FUNCTION_BLOCK Gripper1Ctrl (* Basic Function Block Type *)
  (* Standard: 61499-2 *)
  (* Version 0.0, 3/23/2016, Aalto_IT, nxtControl GmbH, Template *)
  PACKAGE Main;
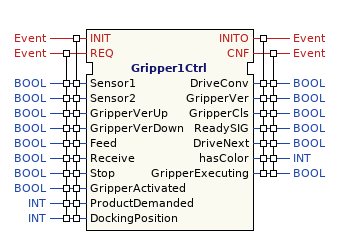
  EVENT_INPUT
    INIT WITH Sensor1, Sensor2, GripperVerUp, GripperVerDown, Feed, Receive, Stop, GripperActivated, ProductDemanded, DockingPosition; (* Initialization Request *)
    REQ WITH Sensor1, Sensor2, GripperVerUp, GripperVerDown, Feed, Receive, Stop, GripperActivated, ProductDemanded, DockingPosition; (* Normal Execution Request *)
  END_EVENT
  EVENT_OUTPUT
    INITO WITH DriveConv, GripperVer, GripperCls, ReadySIG, DriveNext, hasColor, GripperExecuting; (* Initialization Confirm *)
    CNF WITH DriveConv, GripperVer, GripperCls, ReadySIG, DriveNext, hasColor, GripperExecuting; (* Execution Confirmation *)
  END_EVENT
  VAR_INPUT
    Sensor1 : BOOL; (* Input event qualifier *)
    Sensor2 : BOOL;
    GripperVerUp : BOOL;
    GripperVerDown : BOOL;
    Feed : BOOL;
    Receive : BOOL;
    Stop : BOOL;
    GripperActivated : BOOL;
    ProductDemanded : INT;
    DockingPosition : INT;
  END_VAR
  VAR_OUTPUT
    DriveConv : BOOL; (* Output event qualifier *)
    GripperVer : BOOL;
    GripperCls : BOOL;
    ReadySIG : BOOL;
    DriveNext : BOOL;
    hasColor : INT;
    GripperExecuting : BOOL;
  END_VAR
  VAR
    TimeStamp : DATE_AND_TIME;
    SkipWorkCycle : BOOL;
  END_VAR
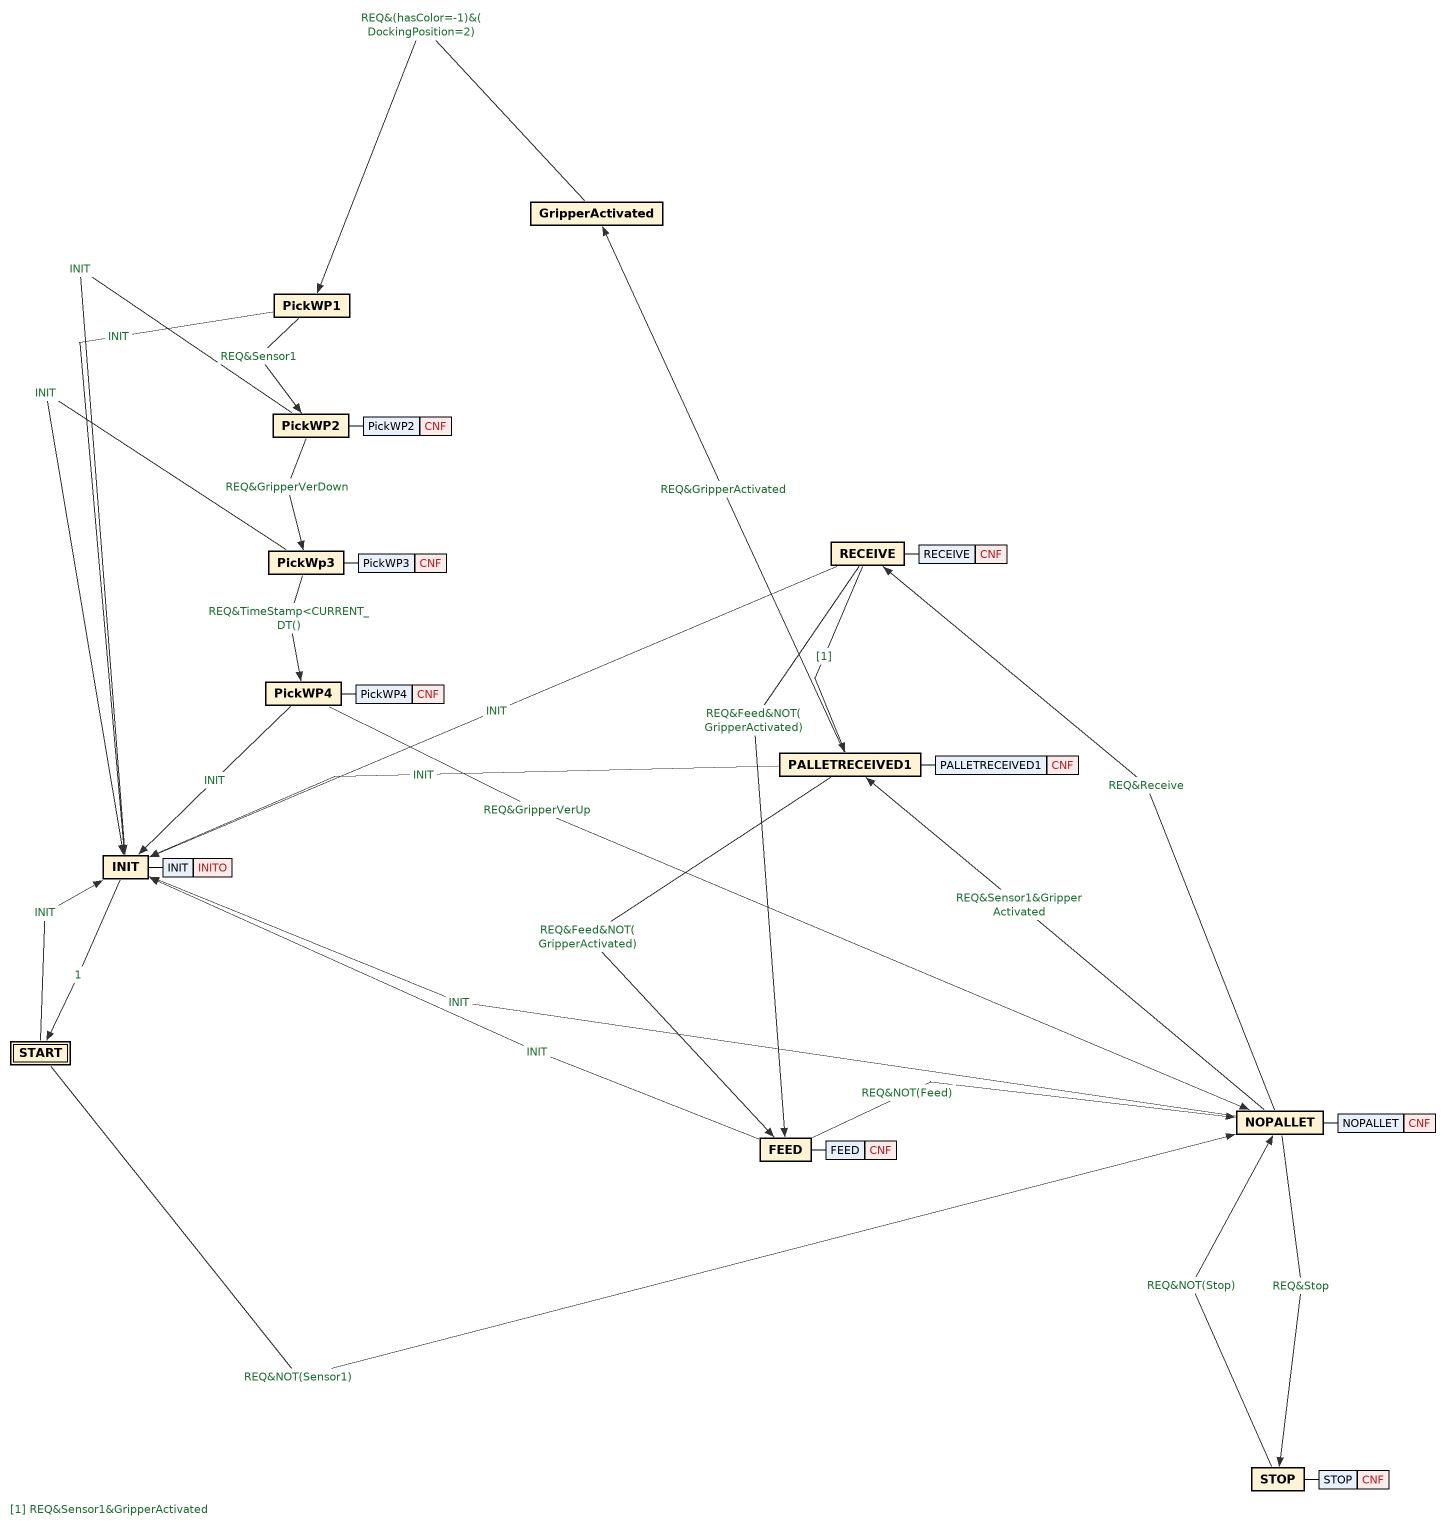
  EC_STATES
    START; (* Initial State *)
    INIT : INIT -> INITO; (* Initialization *)
    NOPALLET : NOPALLET -> CNF;
    PALLETRECEIVED1 : PALLETRECEIVED1 -> CNF;
    FEED : FEED -> CNF;
    RECEIVE : RECEIVE -> CNF;
    STOP : STOP -> CNF;
    GripperActivated;
    PickWP1;
    PickWP2 : PickWP2 -> CNF;
    PickWp3 : PickWP3 -> CNF;
    PickWP4 : PickWP4 -> CNF;
  END_STATES
  EC_TRANSITIONS
    START TO INIT := INIT;
    INIT TO START := 1;
    NOPALLET TO PALLETRECEIVED1 := REQ&Sensor1&GripperActivated;
    PALLETRECEIVED1 TO GripperActivated := REQ&GripperActivated;
    FEED TO NOPALLET := REQ&NOT(Feed);
    PALLETRECEIVED1 TO FEED := REQ&Feed&NOT(GripperActivated);
    NOPALLET TO RECEIVE := REQ&Receive;
    RECEIVE TO PALLETRECEIVED1 := REQ&Sensor1&GripperActivated;
    RECEIVE TO INIT := INIT;
    FEED TO INIT := INIT;
    PALLETRECEIVED1 TO INIT := INIT;
    NOPALLET TO INIT := INIT;
    STOP TO NOPALLET := REQ&NOT(Stop);
    NOPALLET TO STOP := REQ&Stop;
    GripperActivated TO PickWP1 := REQ&(hasColor=-1)&(DockingPosition=2);
    PickWP1 TO PickWP2 := REQ&Sensor1;
    PickWP2 TO PickWp3 := REQ&GripperVerDown;
    PickWp3 TO PickWP4 := REQ&TimeStamp<CURRENT_DT();
    PickWP4 TO NOPALLET := REQ&GripperVerUp;
    PickWP1 TO INIT := INIT;
    PickWP2 TO INIT := INIT;
    PickWp3 TO INIT := INIT;
    PickWP4 TO INIT := INIT;
    START TO NOPALLET := REQ&NOT(Sensor1);
    RECEIVE TO FEED := REQ&Feed&NOT(GripperActivated);
  END_TRANSITIONS
  ALGORITHM INIT IN ST: (* Initialization algorithm *)
DriveConv:=0;
GripperVer:=0;
GripperCls:=0;
DriveNext:=0;
ReadySIG:=1;
hasColor := -1;
GripperExecuting := 0;
// If we dont have any colors
//IF hasColor=-1 THEN
//	GripperCls:=0;
//END_IF;
  END_ALGORITHM
  ALGORITHM REQ IN ST: (* Normally executed algorithm *)
;
  END_ALGORITHM
  ALGORITHM NOPALLET IN ST:
DriveConv:=0;
GripperVer:=0;
//IF (hasColor=-1) THEN
//  GripperCls:=0; //close grippers only if there is no color grasped.
//END_IF;
ReadySIG:=1;
DriveNext:=0;
  END_ALGORITHM
  ALGORITHM PALLETRECEIVED1 IN ST:
DriveConv:=0;
GripperVer:=0;
//IF (hasColor=-1) THEN
//  GripperCls:=0; //close grippers only if there is no color grasped.
//END_IF;
ReadySIG:=0;
DriveNext:=0;
  END_ALGORITHM
  ALGORITHM FEED IN ST:
DriveConv:=1;
GripperVer:=0;
GripperCls:=0;
ReadySIG:=0;
DriveNext:=1;
  END_ALGORITHM
  ALGORITHM RECEIVE IN ST:
DriveConv:=1;
GripperVer:=0;
ReadySIG:=1;
DriveNext:=0;
  END_ALGORITHM
  ALGORITHM STOP IN ST:
DriveConv:=0;
GripperVer:=0;
IF (hasColor=-1) THEN
  GripperCls:=0; //close grippers only if there is no color grasped.
END_IF;
ReadySIG:=0;
DriveNext:=0;
  END_ALGORITHM
  ALGORITHM PickWP2 IN ST:
;
DriveConv:=0;
GripperVer:=1; // Go down...
GripperCls:=0;
ReadySIG:=0;
DriveNext:=0;
  END_ALGORITHM
  ALGORITHM PickWP3 IN ST:
;
DriveConv:=0;
GripperVer:=1;
GripperCls:=1; // close the grippers.
ReadySIG:=0;
DriveNext:=0;
TimeStamp:=ADD_DT_TIME(CURRENT_DT(),T#1.0s); // wait for a moment.
  END_ALGORITHM
  ALGORITHM PickWP4 IN ST:
;
DriveConv:=0;
GripperVer:=0; // Go Up...
GripperCls:=1; // Keep the grippers closed.
ReadySIG:=0;
DriveNext:=0;
hasColor := ProductDemanded; // update the color of the gripper.
DriveNext:=1; // And drive the next conveyor.
  END_ALGORITHM
  ALGORITHM ReceiveWPs IN ST:
;
DriveConv:=1;
GripperVer:=1;
IF (hasColor = -1)THEN
  GripperCls:=0;
END_IF;
DriveNext:=0;
ReadySIG:=0;
//GripperExecuting:=0;
//SkipWorkCycle:=FALSE;
//hasColor := -1;
  END_ALGORITHM
  ALGORITHM ContinueDriving IN ST:
;
DriveConv:=1;
GripperVer:=0;
GripperCls:=0;
DriveNext:=0;
ReadySIG:=1;
  END_ALGORITHM
END_FUNCTION_BLOCK
